{attribute addProperty BoxType "EK1122-0000-0018"}
{attribute addProperty Id "Beckhoff_ER7xxxsub_EK1100EK1100_179A0949162A_0001_ER7041_0002_0024ER7041_5614098424030A_0002_ER7041_0002_0025ER7041_5614098424030A_0003_ER7041_1002_0024ER7041_5614098424030A_0004_ER7041_1002_0025ER7041_5614098424030A_0005_ER7041_2002_0024ER7041_5614098424030A_0006_ER7041_2002_0025ER7041_5614098424030A_0007_ER7041_3002_0021ER7041_E93814AC24030A_0008_ER7041_3002_0022ER7041_E93814AC24030A_0009_ER7342_0002_0020ER7342_5DC6D75238448A_0010_ER7342_0002_0021ER7342_014E044838448A_0011_ER7342_0002_0022ER7342_014E044838448"}
{attribute addProperty CRC "1145641165"}
{attribute addProperty SizeInBites "3088"}
{attribute addProperty SizeInBytes "386"}
TYPE Beckhoff_ER7xxxEK1122_444918CD EXTENDS EK1122_179A0949 :
STRUCT
	{attribute addProperty Name "Beckhoff_ER7xxxsub_EK1100"}
	Beckhoff_ER7xxxsub_EK1100 : EK1100_179A0949;
	{attribute addProperty Name "A_0001_ER7041_0002_0024"}
	A_0001_ER7041_0002_0024 : ER7041_56140984;
	{attribute addProperty Name "A_0002_ER7041_0002_0025"}
	A_0002_ER7041_0002_0025 : ER7041_56140984;
	{attribute addProperty Name "A_0003_ER7041_1002_0024"}
	A_0003_ER7041_1002_0024 : ER7041_56140984;
	{attribute addProperty Name "A_0004_ER7041_1002_0025"}
	A_0004_ER7041_1002_0025 : ER7041_56140984;
	{attribute addProperty Name "A_0005_ER7041_2002_0024"}
	A_0005_ER7041_2002_0024 : ER7041_56140984;
	{attribute addProperty Name "A_0006_ER7041_2002_0025"}
	A_0006_ER7041_2002_0025 : ER7041_56140984;
	{attribute addProperty Name "A_0007_ER7041_3002_0021"}
	A_0007_ER7041_3002_0021 : ER7041_E93814AC;
	{attribute addProperty Name "A_0008_ER7041_3002_0022"}
	A_0008_ER7041_3002_0022 : ER7041_E93814AC;
	{attribute addProperty Name "A_0009_ER7342_0002_0020"}
	A_0009_ER7342_0002_0020 : ER7342_5DC6D752;
	{attribute addProperty Name "A_0010_ER7342_0002_0021"}
	A_0010_ER7342_0002_0021 : ER7342_014E0448;
	{attribute addProperty Name "A_0011_ER7342_0002_0022"}
	A_0011_ER7342_0002_0022 : ER7342_014E0448;
END_STRUCT
END_TYPE

(* stored: Version 1.2.0.0, ProductVersion 3.1.4024.9
   DUT Beckhoff_ER7xxxEK1122_444918CD: Id {61b9cc3b-4f91-4e32-b3f1-e22a9e3c6e84} *)
